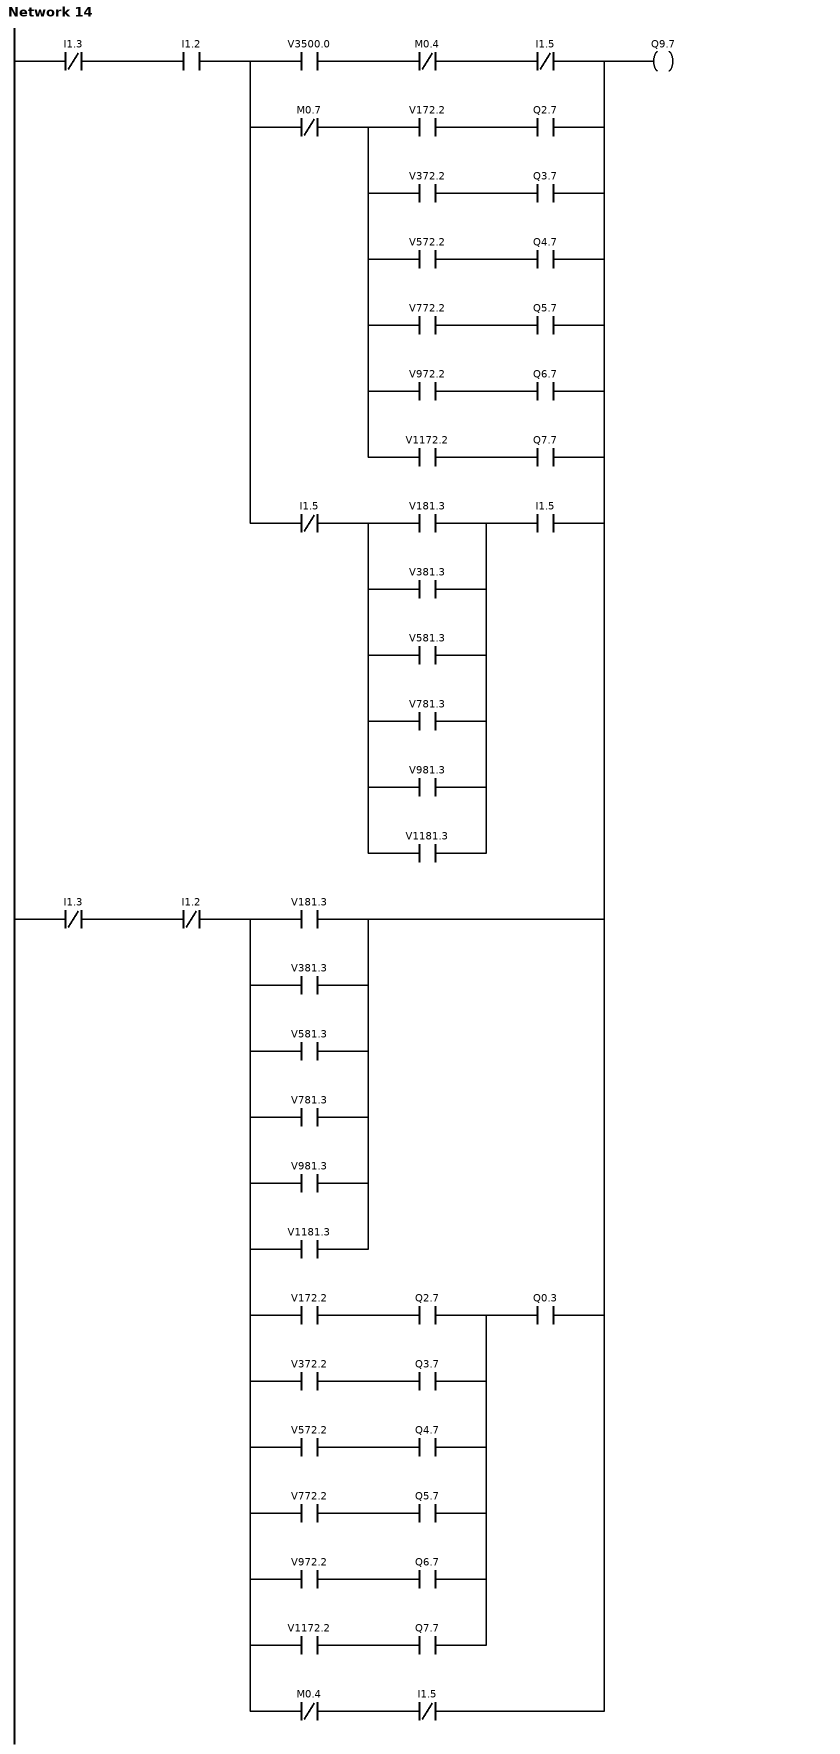
[picture p48: SBR5 networks 14-14]
Network 14
LDN    I1.3
A      I1.2
LD     V3500.0
AN     M0.4
AN     I1.5
LDN    M0.7
LD     V172.2
A      Q2.7
LD     V372.2
A      Q3.7
OLD
LD     V572.2
A      Q4.7
OLD
LD     V772.2
A      Q5.7
OLD
LD     V972.2
A      Q6.7
OLD
LD     V1172.2
A      Q7.7
OLD
ALD
OLD
LDN    I1.5
LD     V181.3
O      V381.3
O      V581.3
O      V781.3
O      V981.3
O      V1181.3
ALD
A      I1.5
OLD
ALD
LDN    I1.3
AN     I1.2
LD     V181.3
O      V381.3
O      V581.3
O      V781.3
O      V981.3
O      V1181.3
LD     V172.2
A      Q2.7
LD     V372.2
A      Q3.7
OLD
LD     V572.2
A      Q4.7
OLD
LD     V772.2
A      Q5.7
OLD
LD     V972.2
A      Q6.7
OLD
LD     V1172.2
A      Q7.7
OLD
A      Q0.3
OLD
LDN    M0.4
AN     I1.5
OLD
ALD
OLD
=      Q9.7
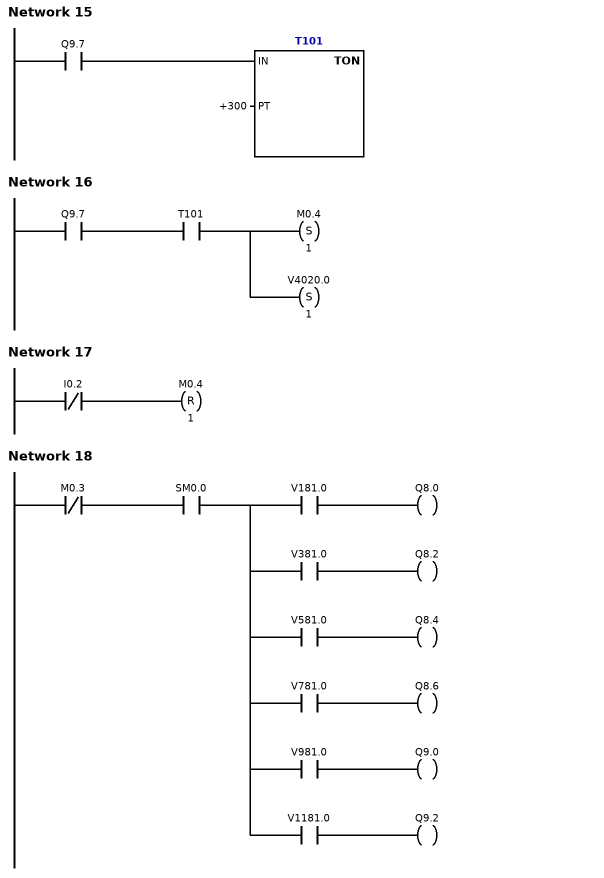
Network 15
LD     Q9.7
TON    T101, +300
Network 16
LD     Q9.7
A      T101
S      M0.4, 1
S      V4020.0, 1
Network 17
LDN    I0.2
R      M0.4, 1
Network 18
LDN    M0.3
A      SM0.0
LPS
A      V181.0
=      Q8.0
LRD
A      V381.0
=      Q8.2
LRD
A      V581.0
=      Q8.4
LRD
A      V781.0
=      Q8.6
LRD
A      V981.0
=      Q9.0
LPP
A      V1181.0
=      Q9.2
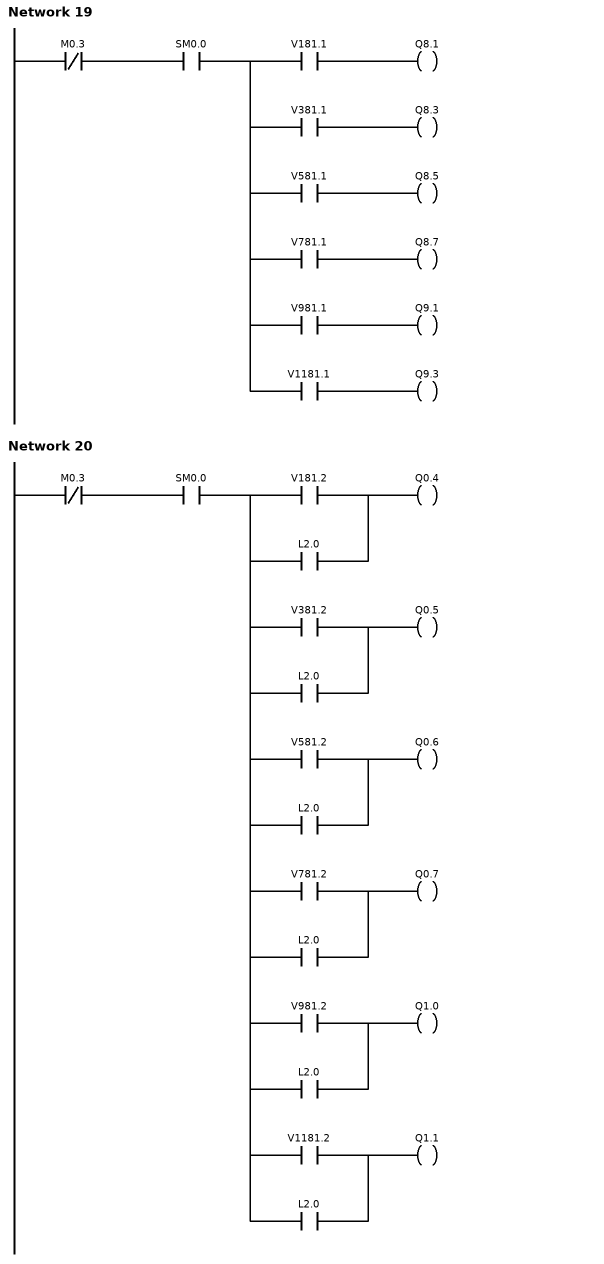
Network 19
LDN    M0.3
A      SM0.0
LPS
A      V181.1
=      Q8.1
LRD
A      V381.1
=      Q8.3
LRD
A      V581.1
=      Q8.5
LRD
A      V781.1
=      Q8.7
LRD
A      V981.1
=      Q9.1
LPP
A      V1181.1
=      Q9.3
Network 20
LDN    M0.3
A      SM0.0
LPS
LD     V181.2
O      L2.0
ALD
=      Q0.4
LRD
LD     V381.2
O      L2.0
ALD
=      Q0.5
LRD
LD     V581.2
O      L2.0
ALD
=      Q0.6
LRD
LD     V781.2
O      L2.0
ALD
=      Q0.7
LRD
LD     V981.2
O      L2.0
ALD
=      Q1.0
LPP
LD     V1181.2
O      L2.0
ALD
=      Q1.1
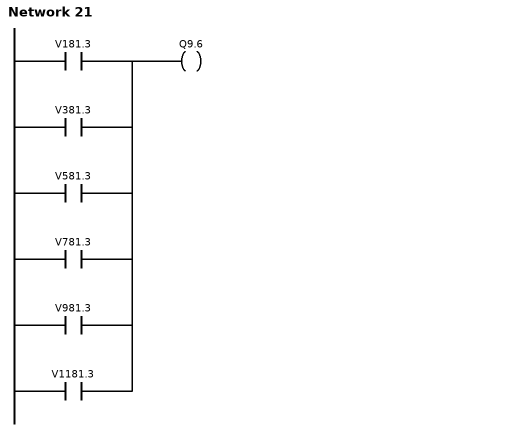
Network 21
LD     V181.3
O      V381.3
O      V581.3
O      V781.3
O      V981.3
O      V1181.3
=      Q9.6
END_SUBROUTINE_BLOCK

SUBROUTINE_BLOCK yz_mc_set:SBR6
TITLE=
BEGIN
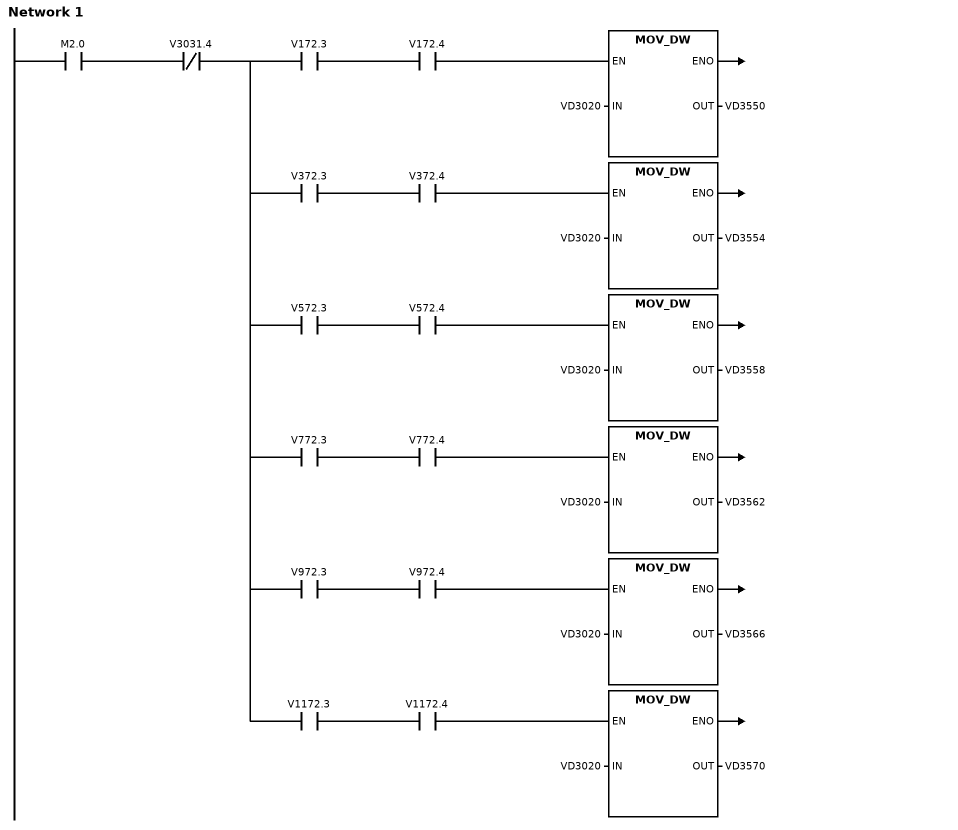
Network 1
LD     M2.0
AN     V3031.4
LPS
A      V172.3
A      V172.4
MOVD   VD3020, VD3550
LRD
A      V372.3
A      V372.4
MOVD   VD3020, VD3554
LRD
A      V572.3
A      V572.4
MOVD   VD3020, VD3558
LRD
A      V772.3
A      V772.4
MOVD   VD3020, VD3562
LRD
A      V972.3
A      V972.4
MOVD   VD3020, VD3566
LPP
A      V1172.3
A      V1172.4
MOVD   VD3020, VD3570
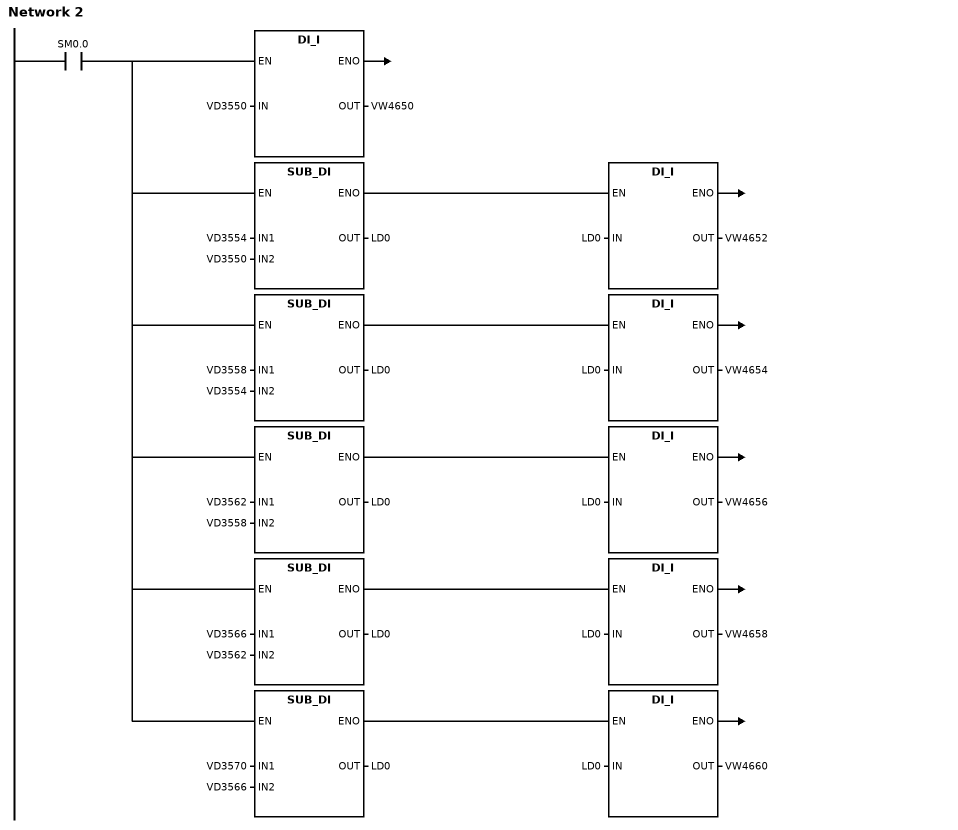
Network 2
LD     SM0.0
LPS
DTI    VD3550, VW4650
MOVD   VD3554, LD0
AENO
-D     VD3550, LD0
AENO
DTI    LD0, VW4652
LRD
MOVD   VD3558, LD0
AENO
-D     VD3554, LD0
AENO
DTI    LD0, VW4654
LRD
MOVD   VD3562, LD0
AENO
-D     VD3558, LD0
AENO
DTI    LD0, VW4656
LRD
MOVD   VD3566, LD0
AENO
-D     VD3562, LD0
AENO
DTI    LD0, VW4658
LPP
MOVD   VD3570, LD0
AENO
-D     VD3566, LD0
AENO
DTI    LD0, VW4660
END_SUBROUTINE_BLOCK

SUBROUTINE_BLOCK STATION_POS:SBR7
TITLE=
BEGIN
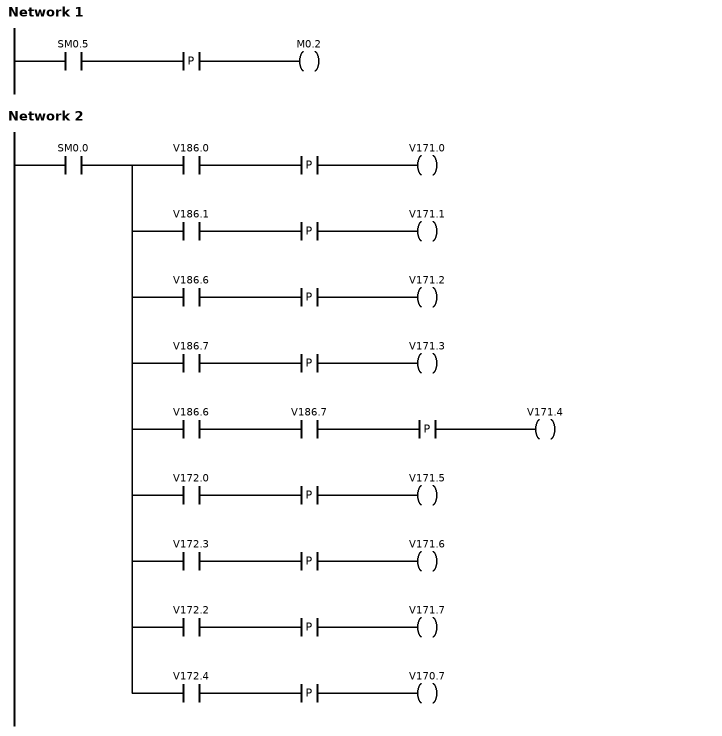
Network 1
LD     SM0.5
EU
=      M0.2
Network 2
LD     SM0.0
LPS
A      V186.0
EU
=      V171.0
LRD
A      V186.1
EU
=      V171.1
LRD
A      V186.6
EU
=      V171.2
LRD
A      V186.7
EU
=      V171.3
LRD
A      V186.6
A      V186.7
EU
=      V171.4
LRD
A      V172.0
EU
=      V171.5
LRD
A      V172.3
EU
=      V171.6
LRD
A      V172.2
EU
=      V171.7
LPP
A      V172.4
EU
=      V170.7
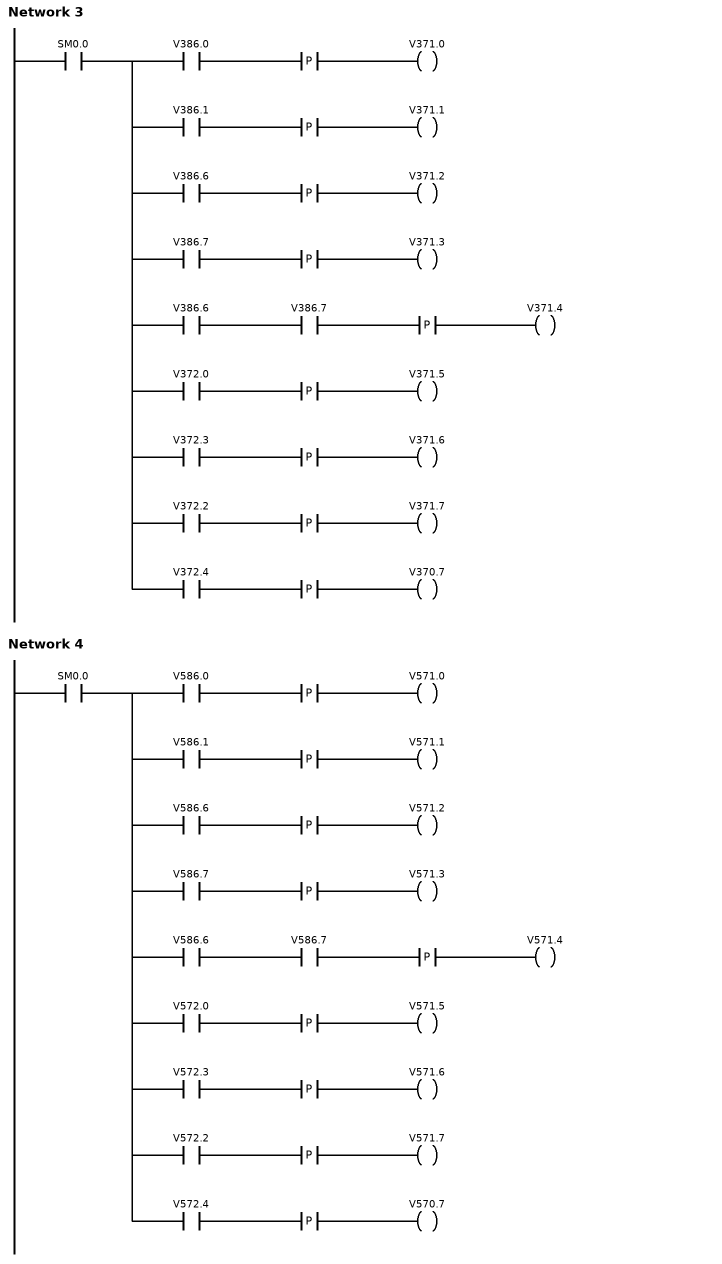
Network 3
LD     SM0.0
LPS
A      V386.0
EU
=      V371.0
LRD
A      V386.1
EU
=      V371.1
LRD
A      V386.6
EU
=      V371.2
LRD
A      V386.7
EU
=      V371.3
LRD
A      V386.6
A      V386.7
EU
=      V371.4
LRD
A      V372.0
EU
=      V371.5
LRD
A      V372.3
EU
=      V371.6
LRD
A      V372.2
EU
=      V371.7
LPP
A      V372.4
EU
=      V370.7
Network 4
LD     SM0.0
LPS
A      V586.0
EU
=      V571.0
LRD
A      V586.1
EU
=      V571.1
LRD
A      V586.6
EU
=      V571.2
LRD
A      V586.7
EU
=      V571.3
LRD
A      V586.6
A      V586.7
EU
=      V571.4
LRD
A      V572.0
EU
=      V571.5
LRD
A      V572.3
EU
=      V571.6
LRD
A      V572.2
EU
=      V571.7
LPP
A      V572.4
EU
=      V570.7
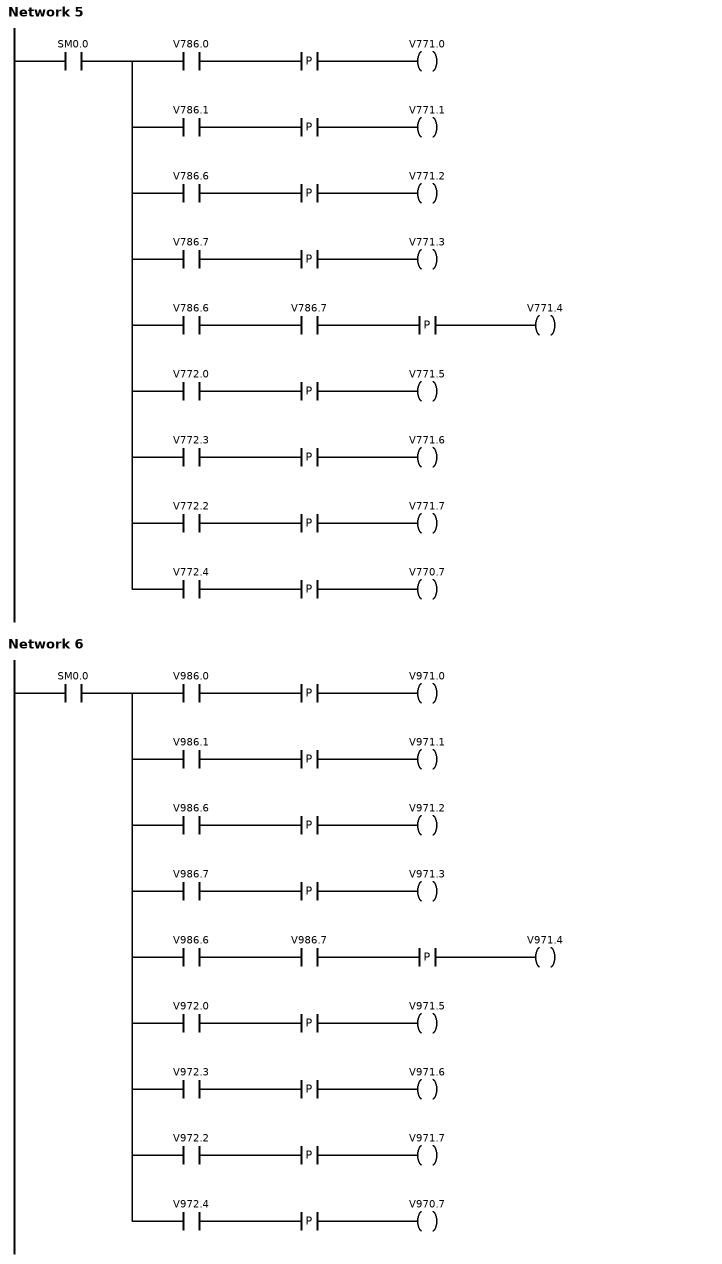
Network 5
LD     SM0.0
LPS
A      V786.0
EU
=      V771.0
LRD
A      V786.1
EU
=      V771.1
LRD
A      V786.6
EU
=      V771.2
LRD
A      V786.7
EU
=      V771.3
LRD
A      V786.6
A      V786.7
EU
=      V771.4
LRD
A      V772.0
EU
=      V771.5
LRD
A      V772.3
EU
=      V771.6
LRD
A      V772.2
EU
=      V771.7
LPP
A      V772.4
EU
=      V770.7
Network 6
LD     SM0.0
LPS
A      V986.0
EU
=      V971.0
LRD
A      V986.1
EU
=      V971.1
LRD
A      V986.6
EU
=      V971.2
LRD
A      V986.7
EU
=      V971.3
LRD
A      V986.6
A      V986.7
EU
=      V971.4
LRD
A      V972.0
EU
=      V971.5
LRD
A      V972.3
EU
=      V971.6
LRD
A      V972.2
EU
=      V971.7
LPP
A      V972.4
EU
=      V970.7
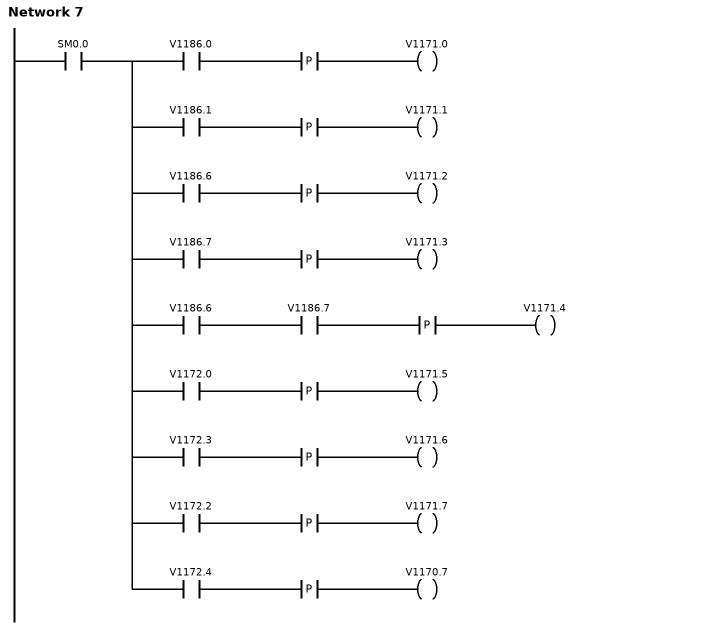
Network 7
LD     SM0.0
LPS
A      V1186.0
EU
=      V1171.0
LRD
A      V1186.1
EU
=      V1171.1
LRD
A      V1186.6
EU
=      V1171.2
LRD
A      V1186.7
EU
=      V1171.3
LRD
A      V1186.6
A      V1186.7
EU
=      V1171.4
LRD
A      V1172.0
EU
=      V1171.5
LRD
A      V1172.3
EU
=      V1171.6
LRD
A      V1172.2
EU
=      V1171.7
LPP
A      V1172.4
EU
=      V1170.7
END_SUBROUTINE_BLOCK

SUBROUTINE_BLOCK AQM_CONTROL:SBR8
TITLE=
BEGIN
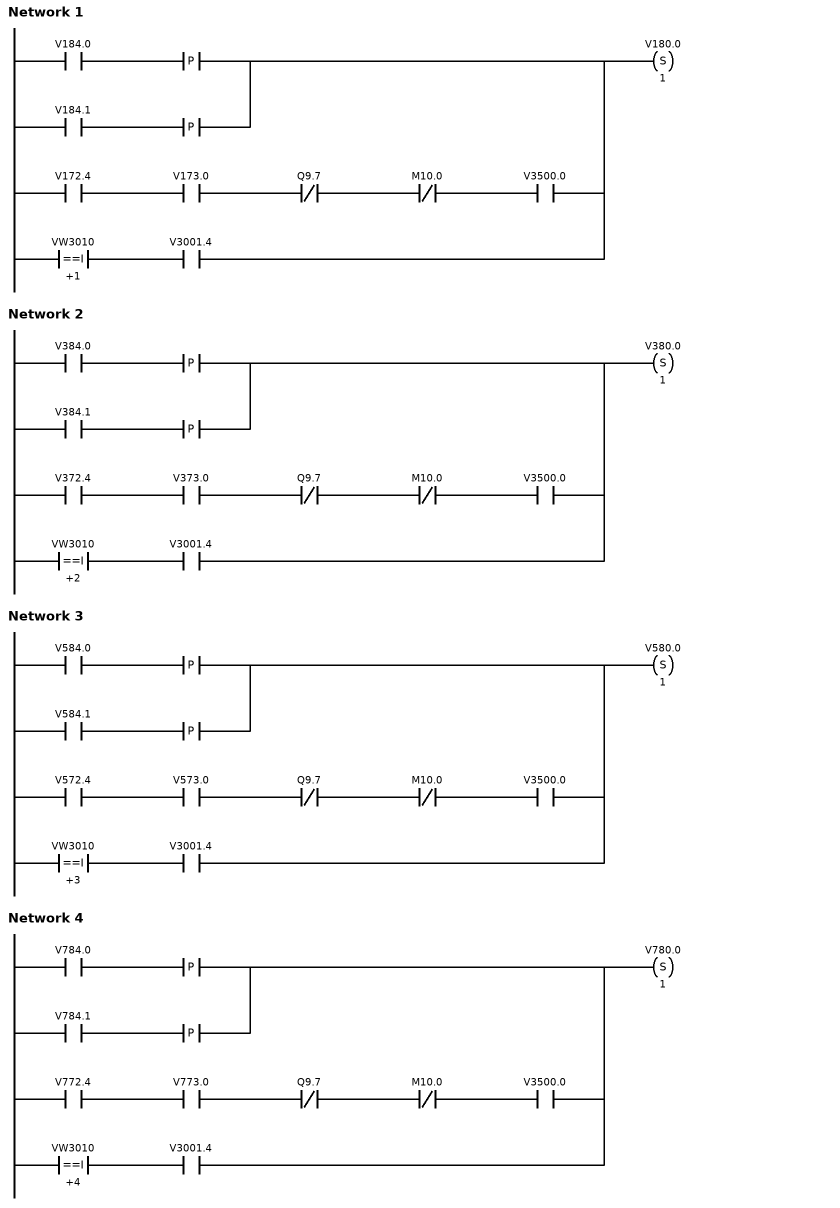
Network 1
LD     V184.0
EU
LD     V184.1
EU
OLD
LD     V172.4
A      V173.0
AN     Q9.7
AN     M10.0
A      V3500.0
OLD
LDW=   VW3010, +1
A      V3001.4
OLD
S      V180.0, 1
Network 2
LD     V384.0
EU
LD     V384.1
EU
OLD
LD     V372.4
A      V373.0
AN     Q9.7
AN     M10.0
A      V3500.0
OLD
LDW=   VW3010, +2
A      V3001.4
OLD
S      V380.0, 1
Network 3
LD     V584.0
EU
LD     V584.1
EU
OLD
LD     V572.4
A      V573.0
AN     Q9.7
AN     M10.0
A      V3500.0
OLD
LDW=   VW3010, +3
A      V3001.4
OLD
S      V580.0, 1
Network 4
LD     V784.0
EU
LD     V784.1
EU
OLD
LD     V772.4
A      V773.0
AN     Q9.7
AN     M10.0
A      V3500.0
OLD
LDW=   VW3010, +4
A      V3001.4
OLD
S      V780.0, 1
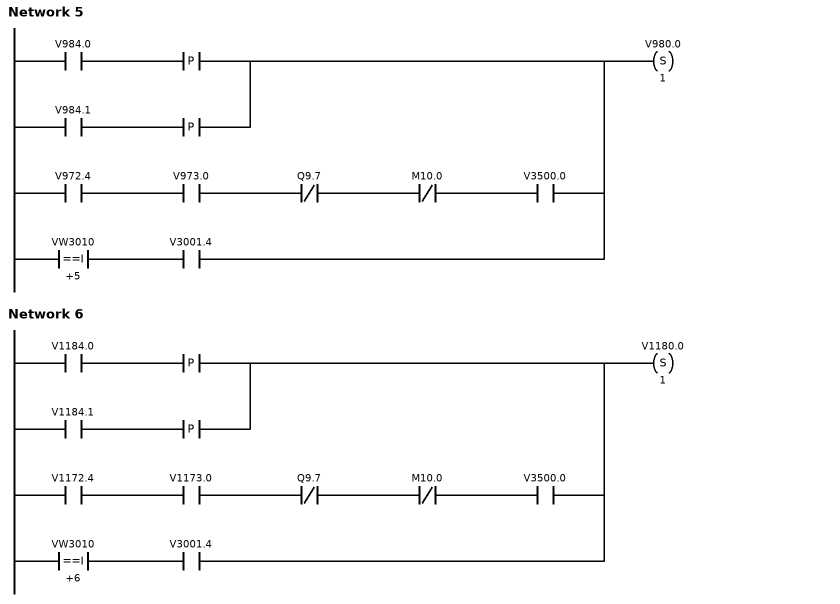
Network 5
LD     V984.0
EU
LD     V984.1
EU
OLD
LD     V972.4
A      V973.0
AN     Q9.7
AN     M10.0
A      V3500.0
OLD
LDW=   VW3010, +5
A      V3001.4
OLD
S      V980.0, 1
Network 6
LD     V1184.0
EU
LD     V1184.1
EU
OLD
LD     V1172.4
A      V1173.0
AN     Q9.7
AN     M10.0
A      V3500.0
OLD
LDW=   VW3010, +6
A      V3001.4
OLD
S      V1180.0, 1
END_SUBROUTINE_BLOCK

SUBROUTINE_BLOCK data_limited:SBR9
TITLE=
BEGIN
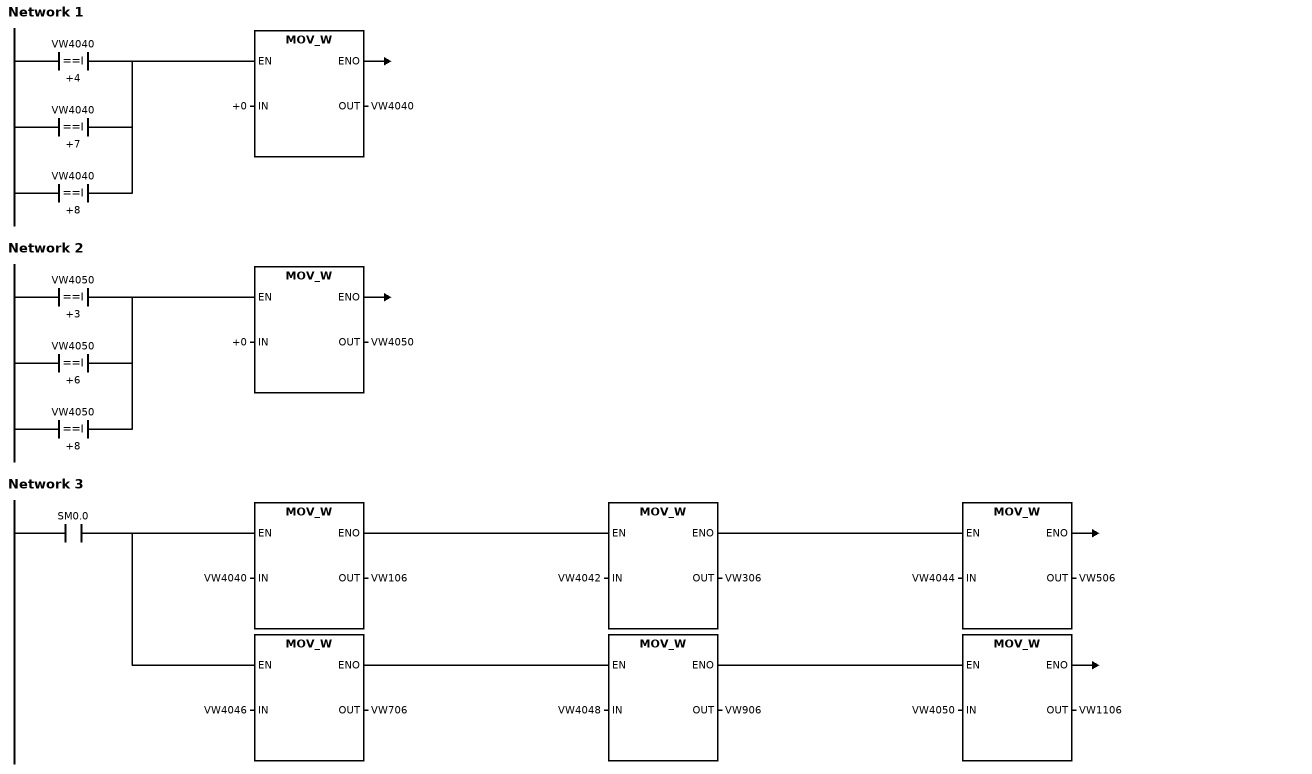
Network 1
LDW=   VW4040, +4
OW=    VW4040, +7
OW=    VW4040, +8
MOVW   +0, VW4040
Network 2
LDW=   VW4050, +3
OW=    VW4050, +6
OW=    VW4050, +8
MOVW   +0, VW4050
Network 3
LD     SM0.0
LPS
MOVW   VW4040, VW106
AENO
MOVW   VW4042, VW306
AENO
MOVW   VW4044, VW506
LPP
MOVW   VW4046, VW706
AENO
MOVW   VW4048, VW906
AENO
MOVW   VW4050, VW1106
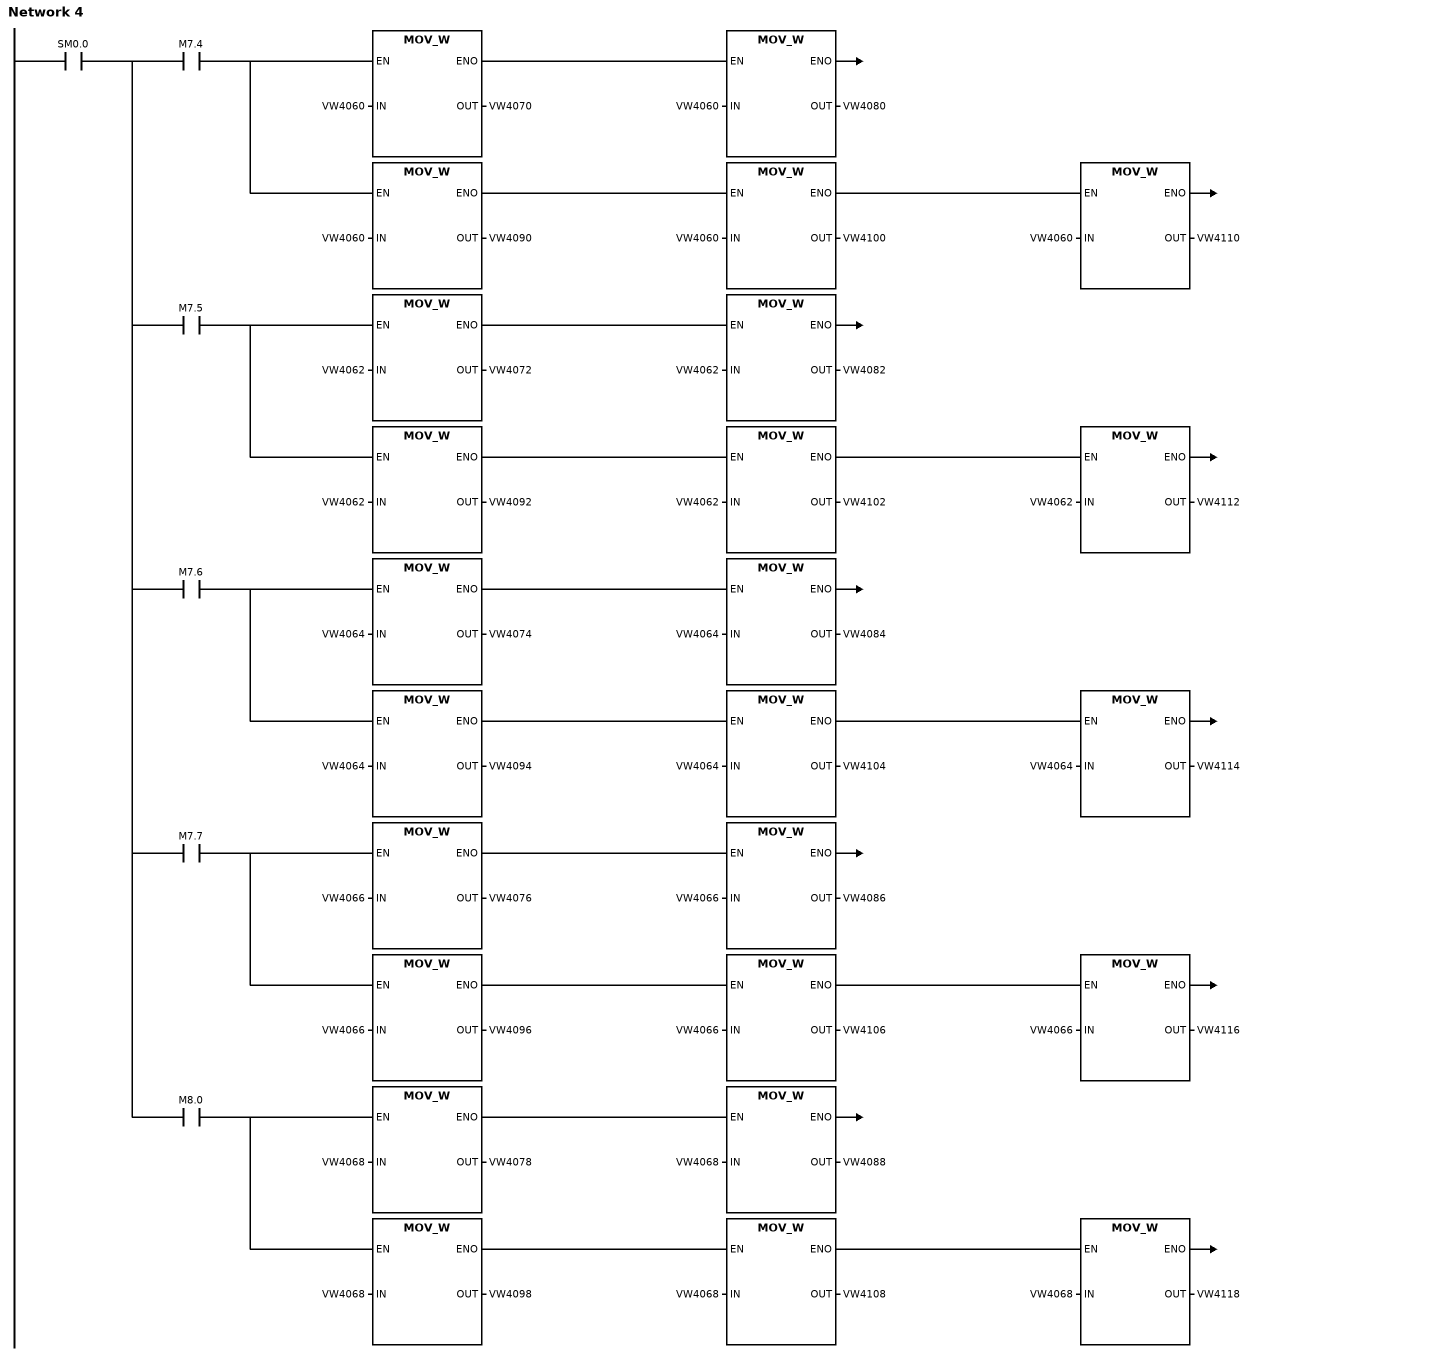
Network 4
LD     SM0.0
LPS
A      M7.4
LPS
MOVW   VW4060, VW4070
AENO
MOVW   VW4060, VW4080
LPP
MOVW   VW4060, VW4090
AENO
MOVW   VW4060, VW4100
AENO
MOVW   VW4060, VW4110
LRD
A      M7.5
LPS
MOVW   VW4062, VW4072
AENO
MOVW   VW4062, VW4082
LPP
MOVW   VW4062, VW4092
AENO
MOVW   VW4062, VW4102
AENO
MOVW   VW4062, VW4112
LRD
A      M7.6
LPS
MOVW   VW4064, VW4074
AENO
MOVW   VW4064, VW4084
LPP
MOVW   VW4064, VW4094
AENO
MOVW   VW4064, VW4104
AENO
MOVW   VW4064, VW4114
LRD
A      M7.7
LPS
MOVW   VW4066, VW4076
AENO
MOVW   VW4066, VW4086
LPP
MOVW   VW4066, VW4096
AENO
MOVW   VW4066, VW4106
AENO
MOVW   VW4066, VW4116
LPP
A      M8.0
LPS
MOVW   VW4068, VW4078
AENO
MOVW   VW4068, VW4088
LPP
MOVW   VW4068, VW4098
AENO
MOVW   VW4068, VW4108
AENO
MOVW   VW4068, VW4118
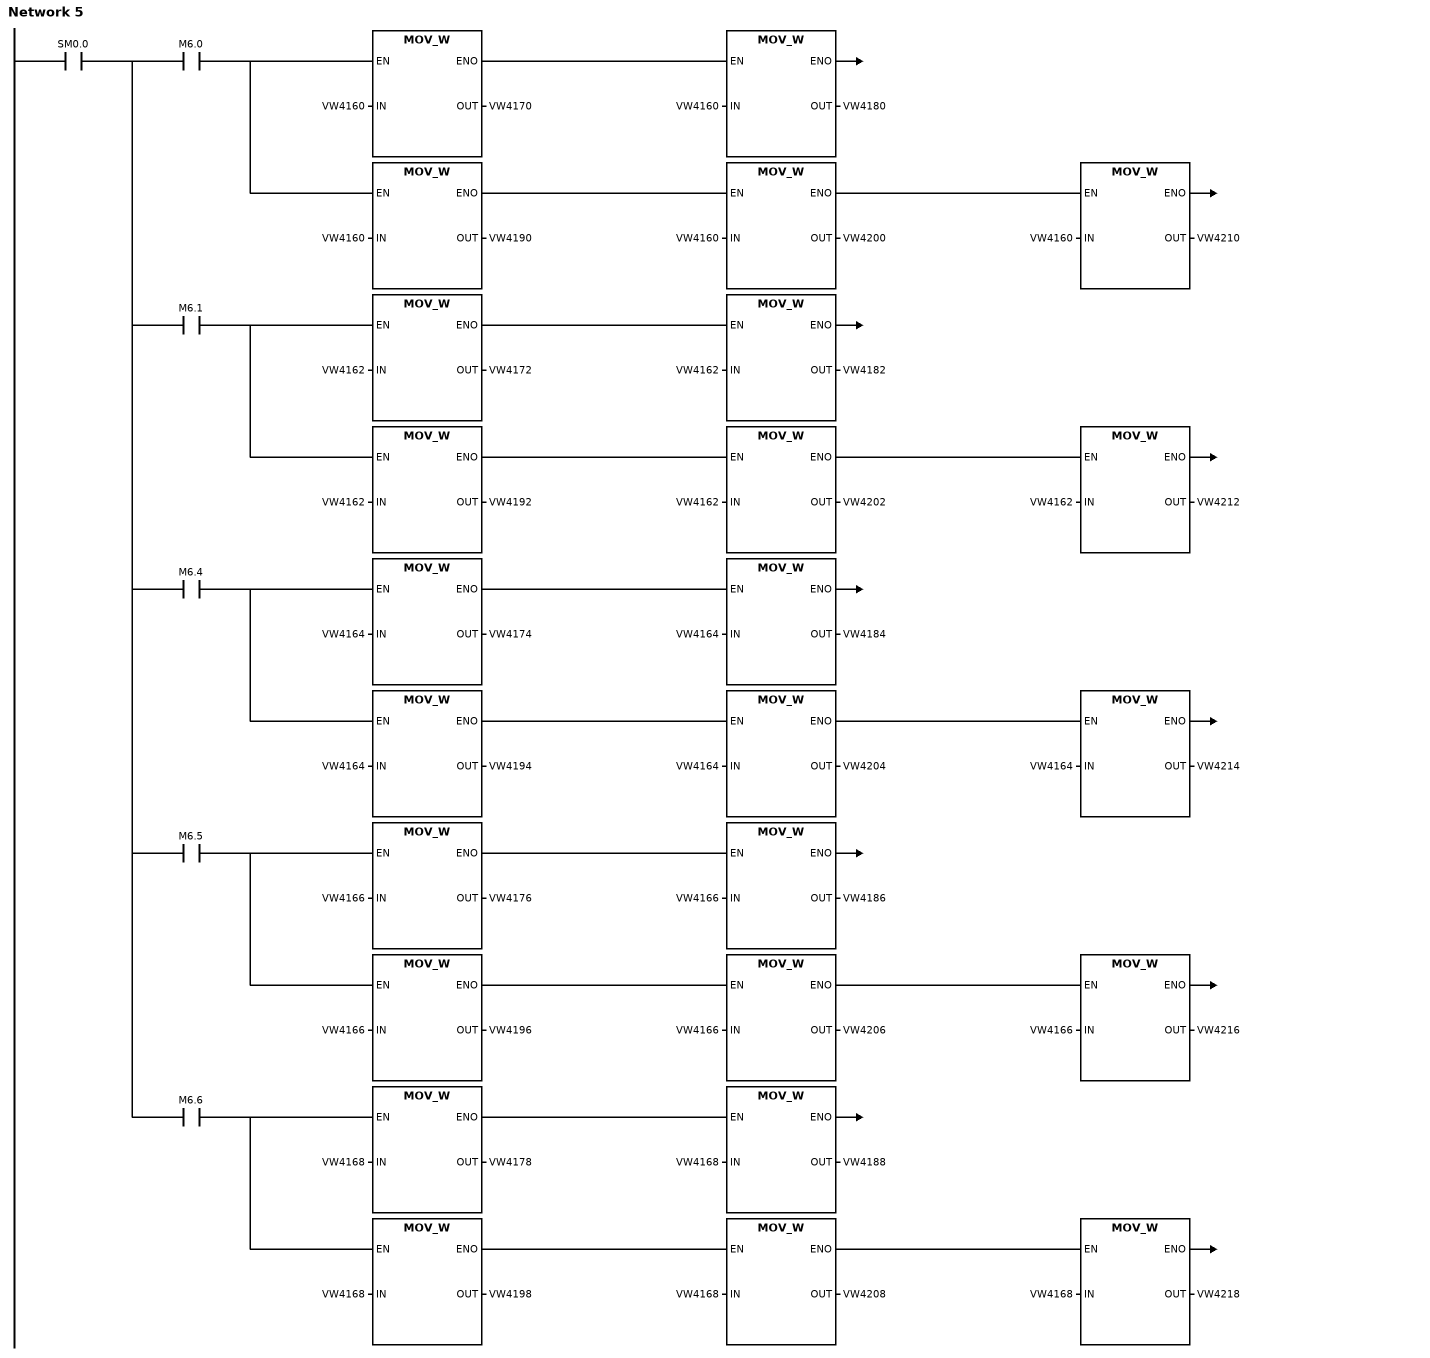
Network 5
LD     SM0.0
LPS
A      M6.0
LPS
MOVW   VW4160, VW4170
AENO
MOVW   VW4160, VW4180
LPP
MOVW   VW4160, VW4190
AENO
MOVW   VW4160, VW4200
AENO
MOVW   VW4160, VW4210
LRD
A      M6.1
LPS
MOVW   VW4162, VW4172
AENO
MOVW   VW4162, VW4182
LPP
MOVW   VW4162, VW4192
AENO
MOVW   VW4162, VW4202
AENO
MOVW   VW4162, VW4212
LRD
A      M6.4
LPS
MOVW   VW4164, VW4174
AENO
MOVW   VW4164, VW4184
LPP
MOVW   VW4164, VW4194
AENO
MOVW   VW4164, VW4204
AENO
MOVW   VW4164, VW4214
LRD
A      M6.5
LPS
MOVW   VW4166, VW4176
AENO
MOVW   VW4166, VW4186
LPP
MOVW   VW4166, VW4196
AENO
MOVW   VW4166, VW4206
AENO
MOVW   VW4166, VW4216
LPP
A      M6.6
LPS
MOVW   VW4168, VW4178
AENO
MOVW   VW4168, VW4188
LPP
MOVW   VW4168, VW4198
AENO
MOVW   VW4168, VW4208
AENO
MOVW   VW4168, VW4218
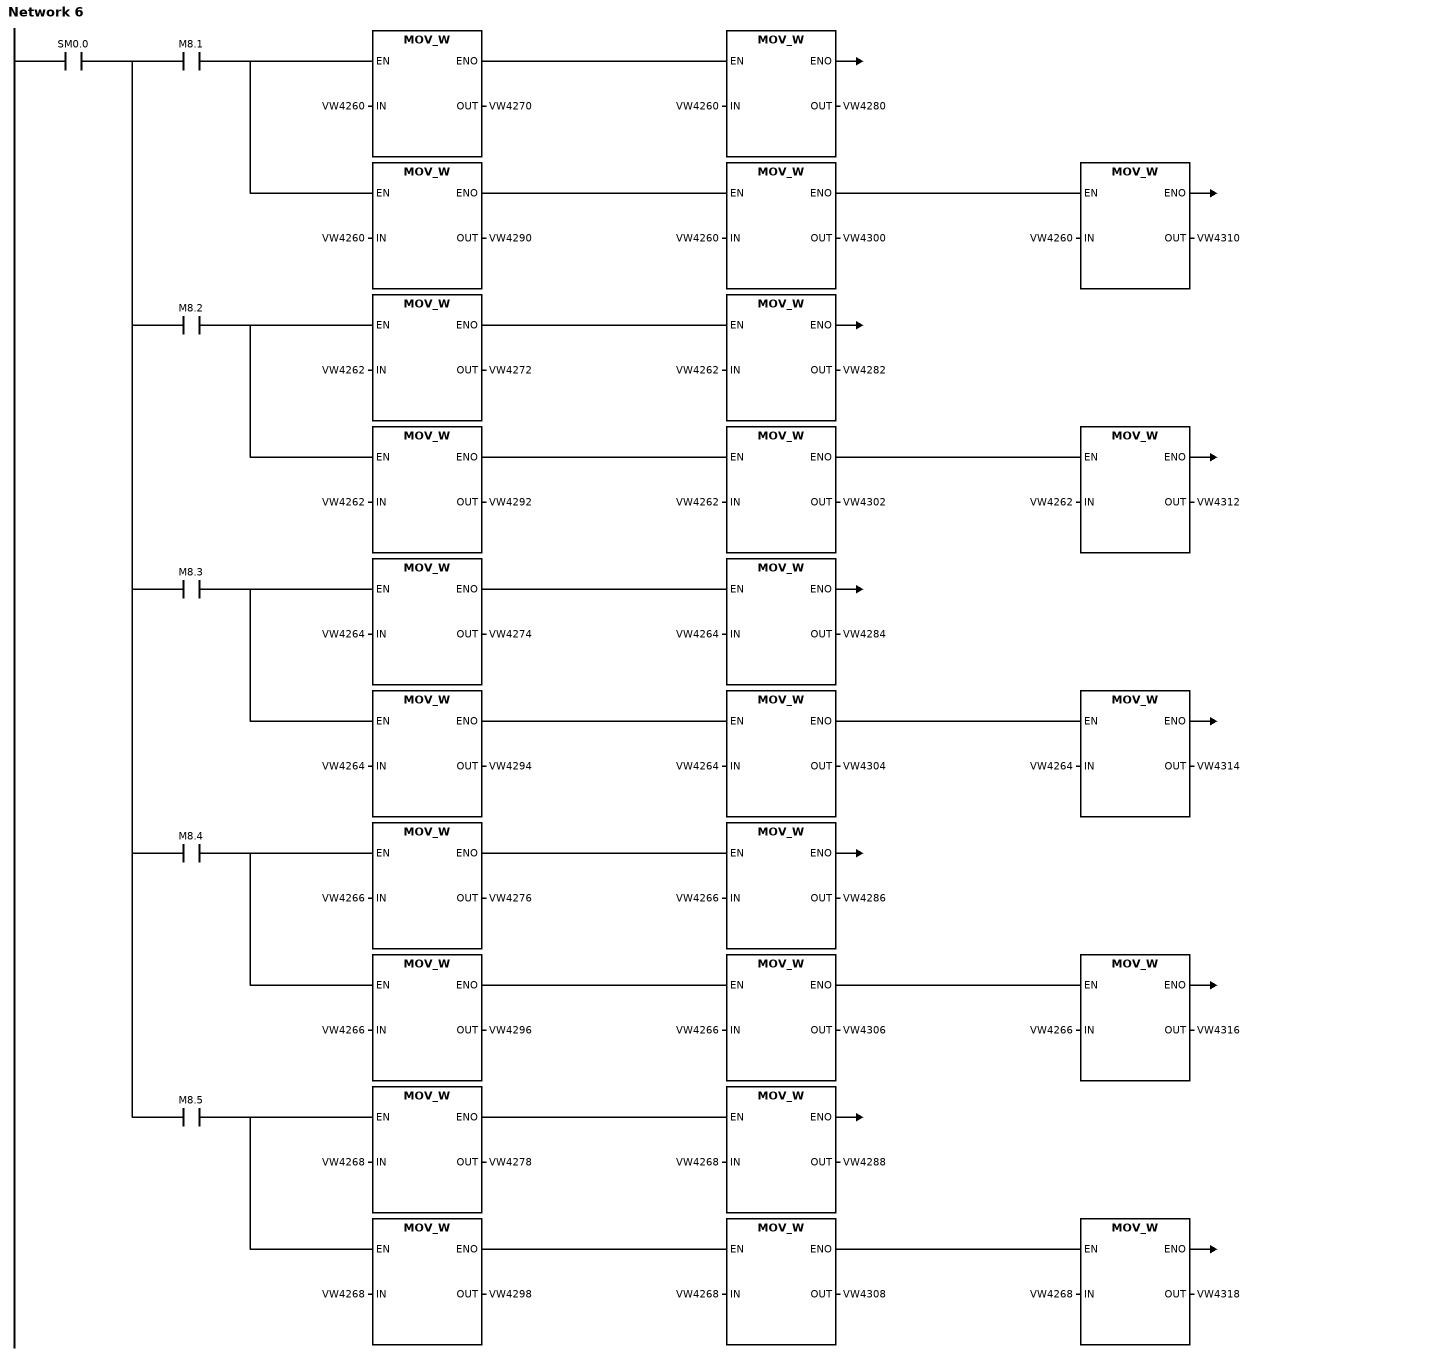
Network 6
LD     SM0.0
LPS
A      M8.1
LPS
MOVW   VW4260, VW4270
AENO
MOVW   VW4260, VW4280
LPP
MOVW   VW4260, VW4290
AENO
MOVW   VW4260, VW4300
AENO
MOVW   VW4260, VW4310
LRD
A      M8.2
LPS
MOVW   VW4262, VW4272
AENO
MOVW   VW4262, VW4282
LPP
MOVW   VW4262, VW4292
AENO
MOVW   VW4262, VW4302
AENO
MOVW   VW4262, VW4312
LRD
A      M8.3
LPS
MOVW   VW4264, VW4274
AENO
MOVW   VW4264, VW4284
LPP
MOVW   VW4264, VW4294
AENO
MOVW   VW4264, VW4304
AENO
MOVW   VW4264, VW4314
LRD
A      M8.4
LPS
MOVW   VW4266, VW4276
AENO
MOVW   VW4266, VW4286
LPP
MOVW   VW4266, VW4296
AENO
MOVW   VW4266, VW4306
AENO
MOVW   VW4266, VW4316
LPP
A      M8.5
LPS
MOVW   VW4268, VW4278
AENO
MOVW   VW4268, VW4288
LPP
MOVW   VW4268, VW4298
AENO
MOVW   VW4268, VW4308
AENO
MOVW   VW4268, VW4318
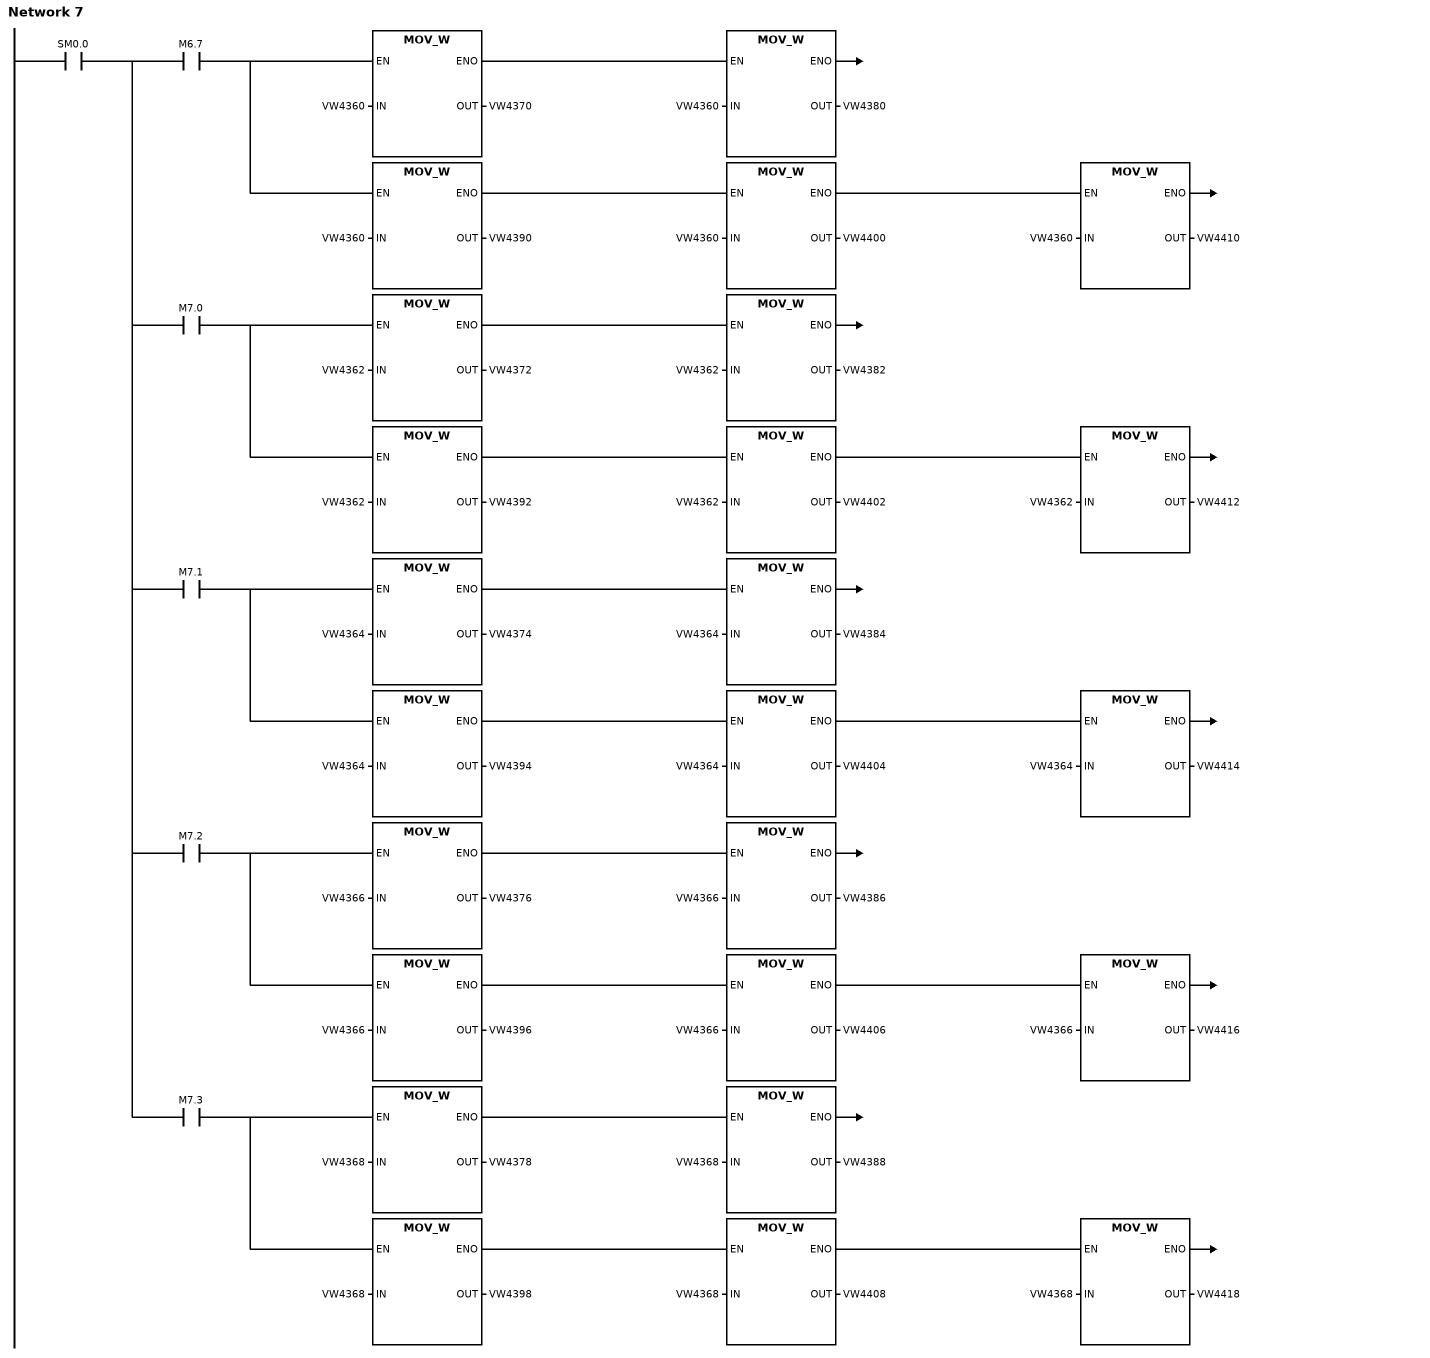
Network 7
LD     SM0.0
LPS
A      M6.7
LPS
MOVW   VW4360, VW4370
AENO
MOVW   VW4360, VW4380
LPP
MOVW   VW4360, VW4390
AENO
MOVW   VW4360, VW4400
AENO
MOVW   VW4360, VW4410
LRD
A      M7.0
LPS
MOVW   VW4362, VW4372
AENO
MOVW   VW4362, VW4382
LPP
MOVW   VW4362, VW4392
AENO
MOVW   VW4362, VW4402
AENO
MOVW   VW4362, VW4412
LRD
A      M7.1
LPS
MOVW   VW4364, VW4374
AENO
MOVW   VW4364, VW4384
LPP
MOVW   VW4364, VW4394
AENO
MOVW   VW4364, VW4404
AENO
MOVW   VW4364, VW4414
LRD
A      M7.2
LPS
MOVW   VW4366, VW4376
AENO
MOVW   VW4366, VW4386
LPP
MOVW   VW4366, VW4396
AENO
MOVW   VW4366, VW4406
AENO
MOVW   VW4366, VW4416
LPP
A      M7.3
LPS
MOVW   VW4368, VW4378
AENO
MOVW   VW4368, VW4388
LPP
MOVW   VW4368, VW4398
AENO
MOVW   VW4368, VW4408
AENO
MOVW   VW4368, VW4418
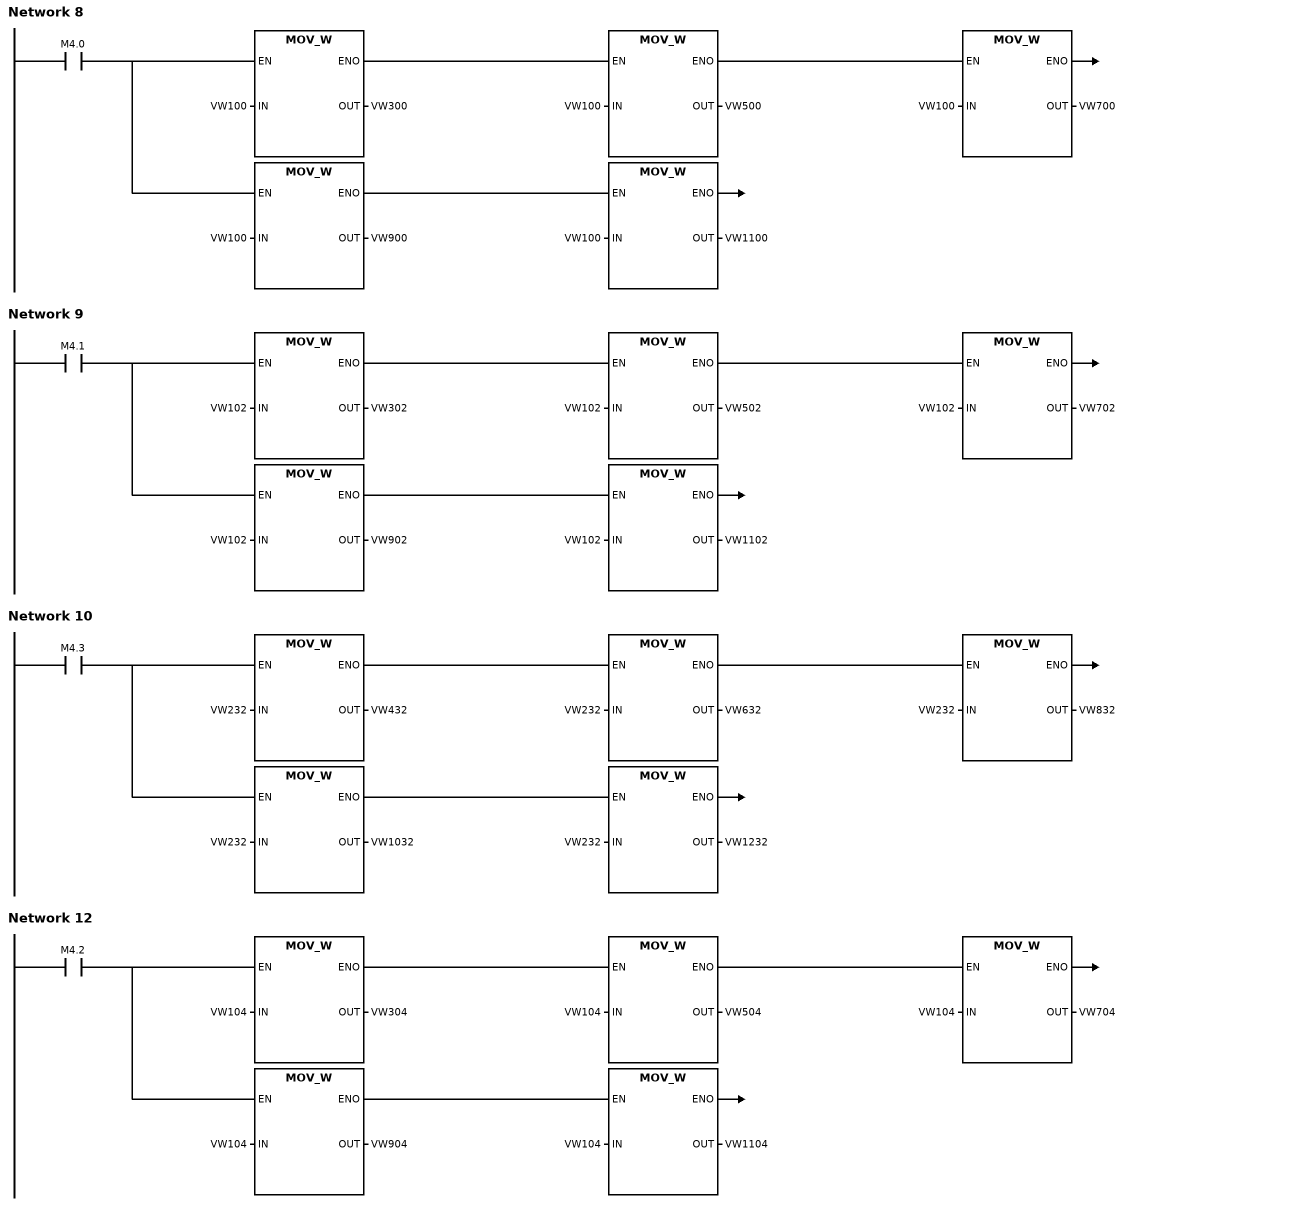
Network 8
LD     M4.0
LPS
MOVW   VW100, VW300
AENO
MOVW   VW100, VW500
AENO
MOVW   VW100, VW700
LPP
MOVW   VW100, VW900
AENO
MOVW   VW100, VW1100
Network 9
LD     M4.1
LPS
MOVW   VW102, VW302
AENO
MOVW   VW102, VW502
AENO
MOVW   VW102, VW702
LPP
MOVW   VW102, VW902
AENO
MOVW   VW102, VW1102
Network 10
LD     M4.3
LPS
MOVW   VW232, VW432
AENO
MOVW   VW232, VW632
AENO
MOVW   VW232, VW832
LPP
MOVW   VW232, VW1032
AENO
MOVW   VW232, VW1232
Network 12
LD     M4.2
LPS
MOVW   VW104, VW304
AENO
MOVW   VW104, VW504
AENO
MOVW   VW104, VW704
LPP
MOVW   VW104, VW904
AENO
MOVW   VW104, VW1104
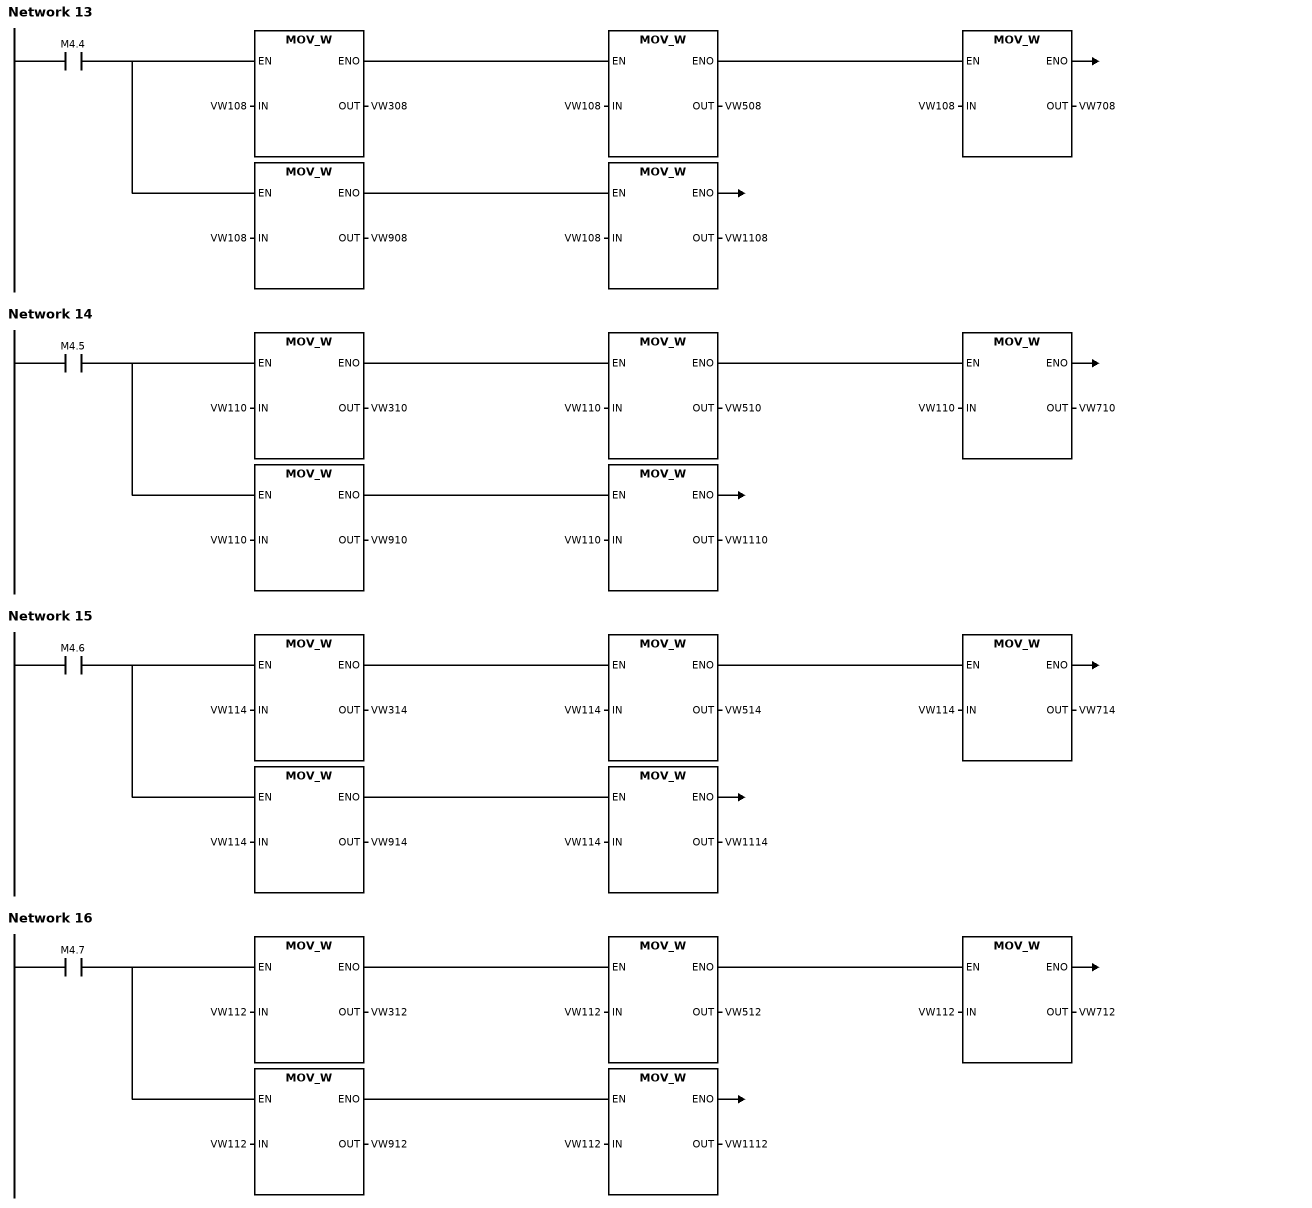
Network 13
LD     M4.4
LPS
MOVW   VW108, VW308
AENO
MOVW   VW108, VW508
AENO
MOVW   VW108, VW708
LPP
MOVW   VW108, VW908
AENO
MOVW   VW108, VW1108
Network 14
LD     M4.5
LPS
MOVW   VW110, VW310
AENO
MOVW   VW110, VW510
AENO
MOVW   VW110, VW710
LPP
MOVW   VW110, VW910
AENO
MOVW   VW110, VW1110
Network 15
LD     M4.6
LPS
MOVW   VW114, VW314
AENO
MOVW   VW114, VW514
AENO
MOVW   VW114, VW714
LPP
MOVW   VW114, VW914
AENO
MOVW   VW114, VW1114
Network 16
LD     M4.7
LPS
MOVW   VW112, VW312
AENO
MOVW   VW112, VW512
AENO
MOVW   VW112, VW712
LPP
MOVW   VW112, VW912
AENO
MOVW   VW112, VW1112
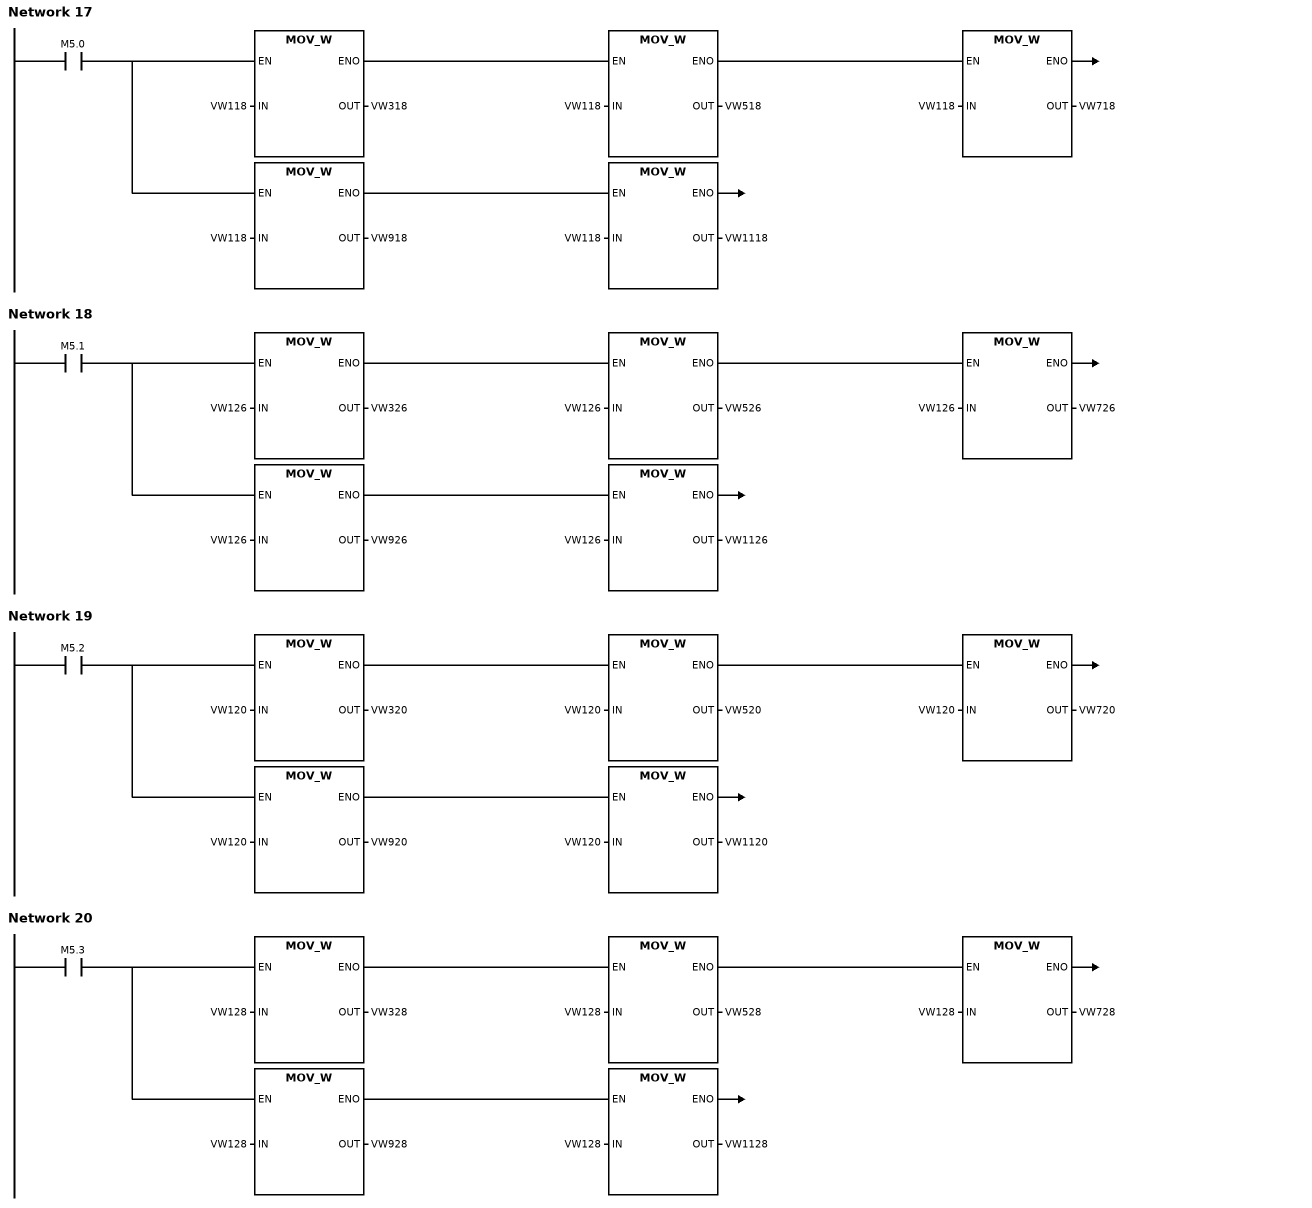
Network 17
LD     M5.0
LPS
MOVW   VW118, VW318
AENO
MOVW   VW118, VW518
AENO
MOVW   VW118, VW718
LPP
MOVW   VW118, VW918
AENO
MOVW   VW118, VW1118
Network 18
LD     M5.1
LPS
MOVW   VW126, VW326
AENO
MOVW   VW126, VW526
AENO
MOVW   VW126, VW726
LPP
MOVW   VW126, VW926
AENO
MOVW   VW126, VW1126
Network 19
LD     M5.2
LPS
MOVW   VW120, VW320
AENO
MOVW   VW120, VW520
AENO
MOVW   VW120, VW720
LPP
MOVW   VW120, VW920
AENO
MOVW   VW120, VW1120
Network 20
LD     M5.3
LPS
MOVW   VW128, VW328
AENO
MOVW   VW128, VW528
AENO
MOVW   VW128, VW728
LPP
MOVW   VW128, VW928
AENO
MOVW   VW128, VW1128
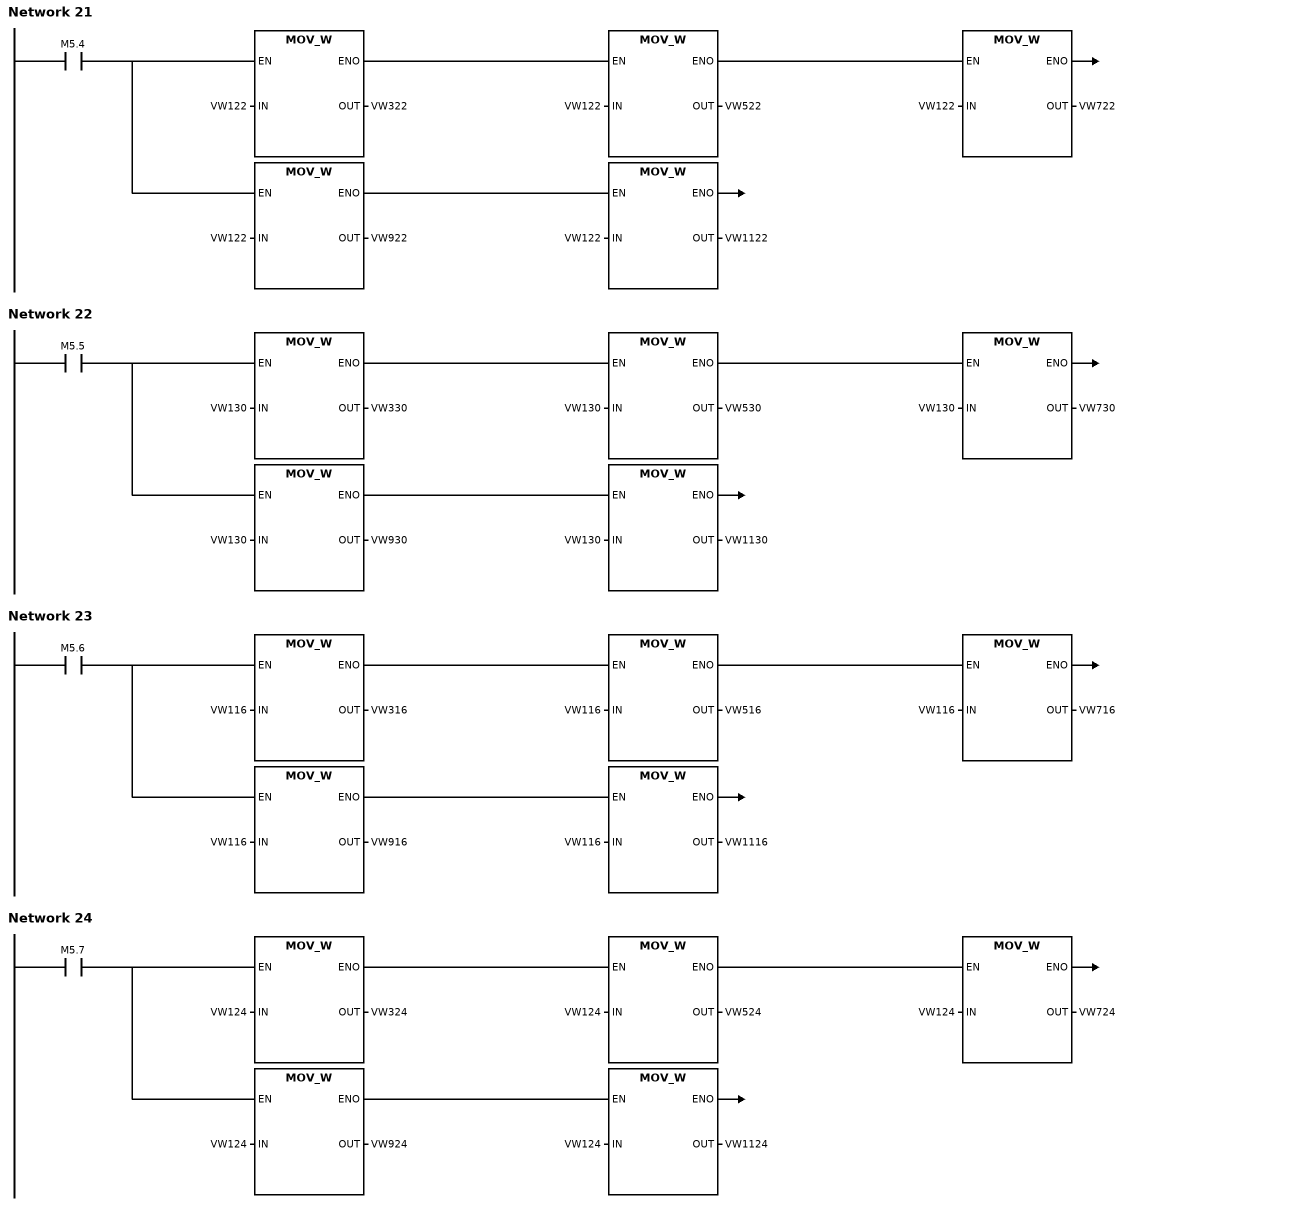
Network 21
LD     M5.4
LPS
MOVW   VW122, VW322
AENO
MOVW   VW122, VW522
AENO
MOVW   VW122, VW722
LPP
MOVW   VW122, VW922
AENO
MOVW   VW122, VW1122
Network 22
LD     M5.5
LPS
MOVW   VW130, VW330
AENO
MOVW   VW130, VW530
AENO
MOVW   VW130, VW730
LPP
MOVW   VW130, VW930
AENO
MOVW   VW130, VW1130
Network 23
LD     M5.6
LPS
MOVW   VW116, VW316
AENO
MOVW   VW116, VW516
AENO
MOVW   VW116, VW716
LPP
MOVW   VW116, VW916
AENO
MOVW   VW116, VW1116
Network 24
LD     M5.7
LPS
MOVW   VW124, VW324
AENO
MOVW   VW124, VW524
AENO
MOVW   VW124, VW724
LPP
MOVW   VW124, VW924
AENO
MOVW   VW124, VW1124
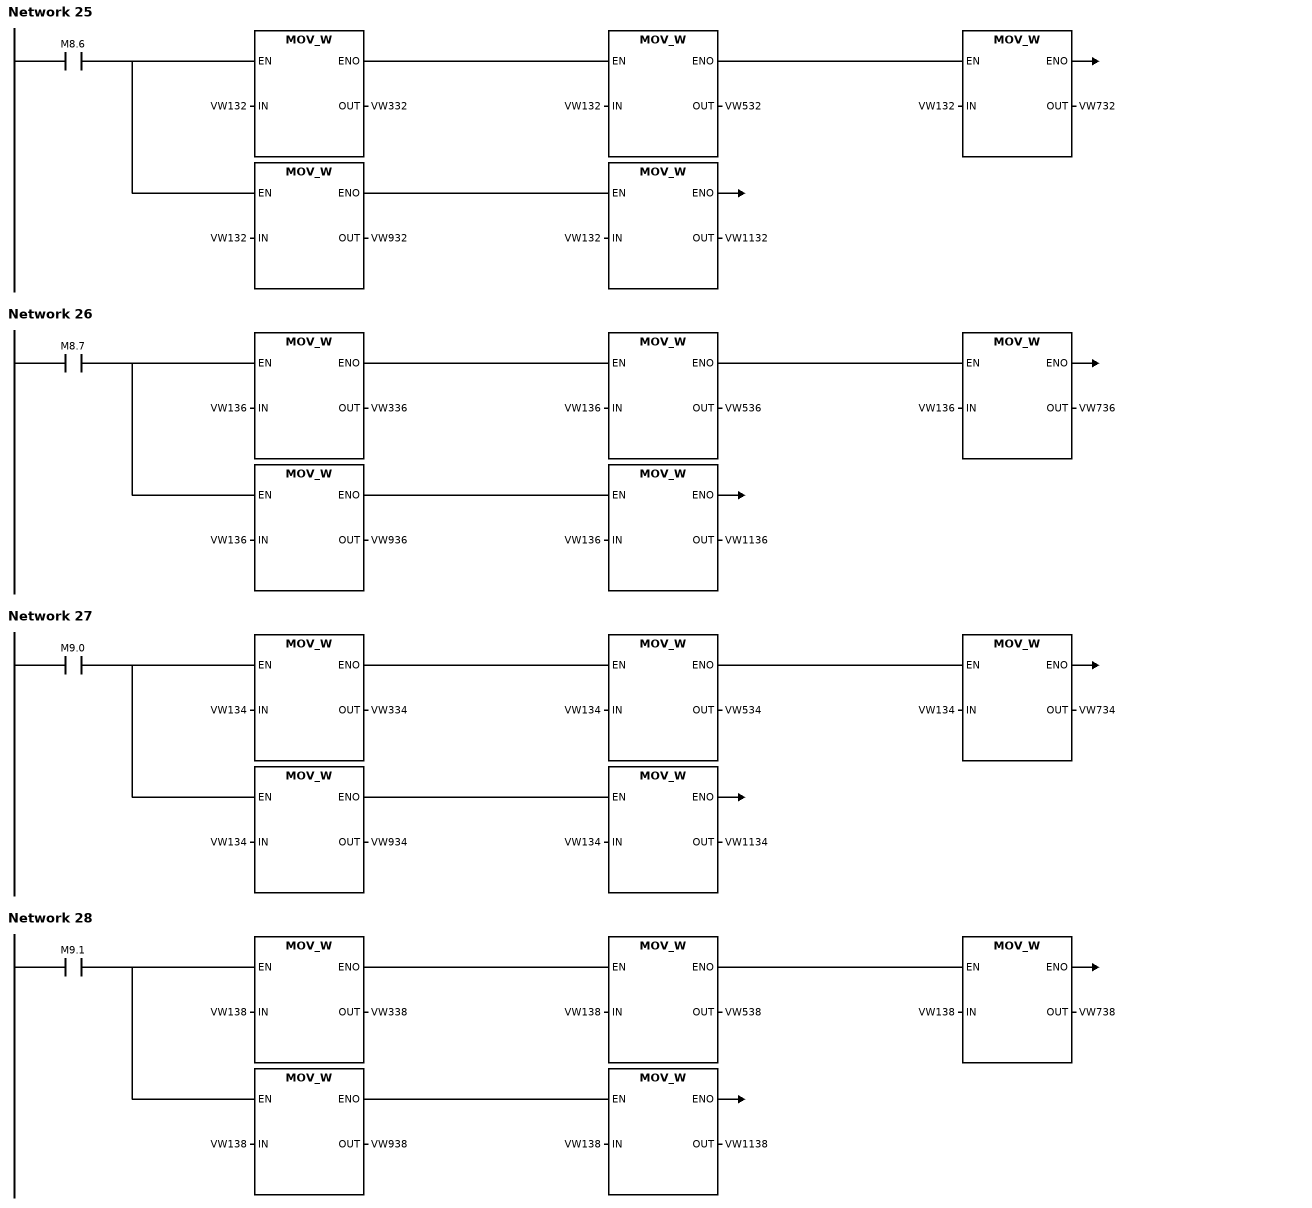
Network 25
LD     M8.6
LPS
MOVW   VW132, VW332
AENO
MOVW   VW132, VW532
AENO
MOVW   VW132, VW732
LPP
MOVW   VW132, VW932
AENO
MOVW   VW132, VW1132
Network 26
LD     M8.7
LPS
MOVW   VW136, VW336
AENO
MOVW   VW136, VW536
AENO
MOVW   VW136, VW736
LPP
MOVW   VW136, VW936
AENO
MOVW   VW136, VW1136
Network 27
LD     M9.0
LPS
MOVW   VW134, VW334
AENO
MOVW   VW134, VW534
AENO
MOVW   VW134, VW734
LPP
MOVW   VW134, VW934
AENO
MOVW   VW134, VW1134
Network 28
LD     M9.1
LPS
MOVW   VW138, VW338
AENO
MOVW   VW138, VW538
AENO
MOVW   VW138, VW738
LPP
MOVW   VW138, VW938
AENO
MOVW   VW138, VW1138
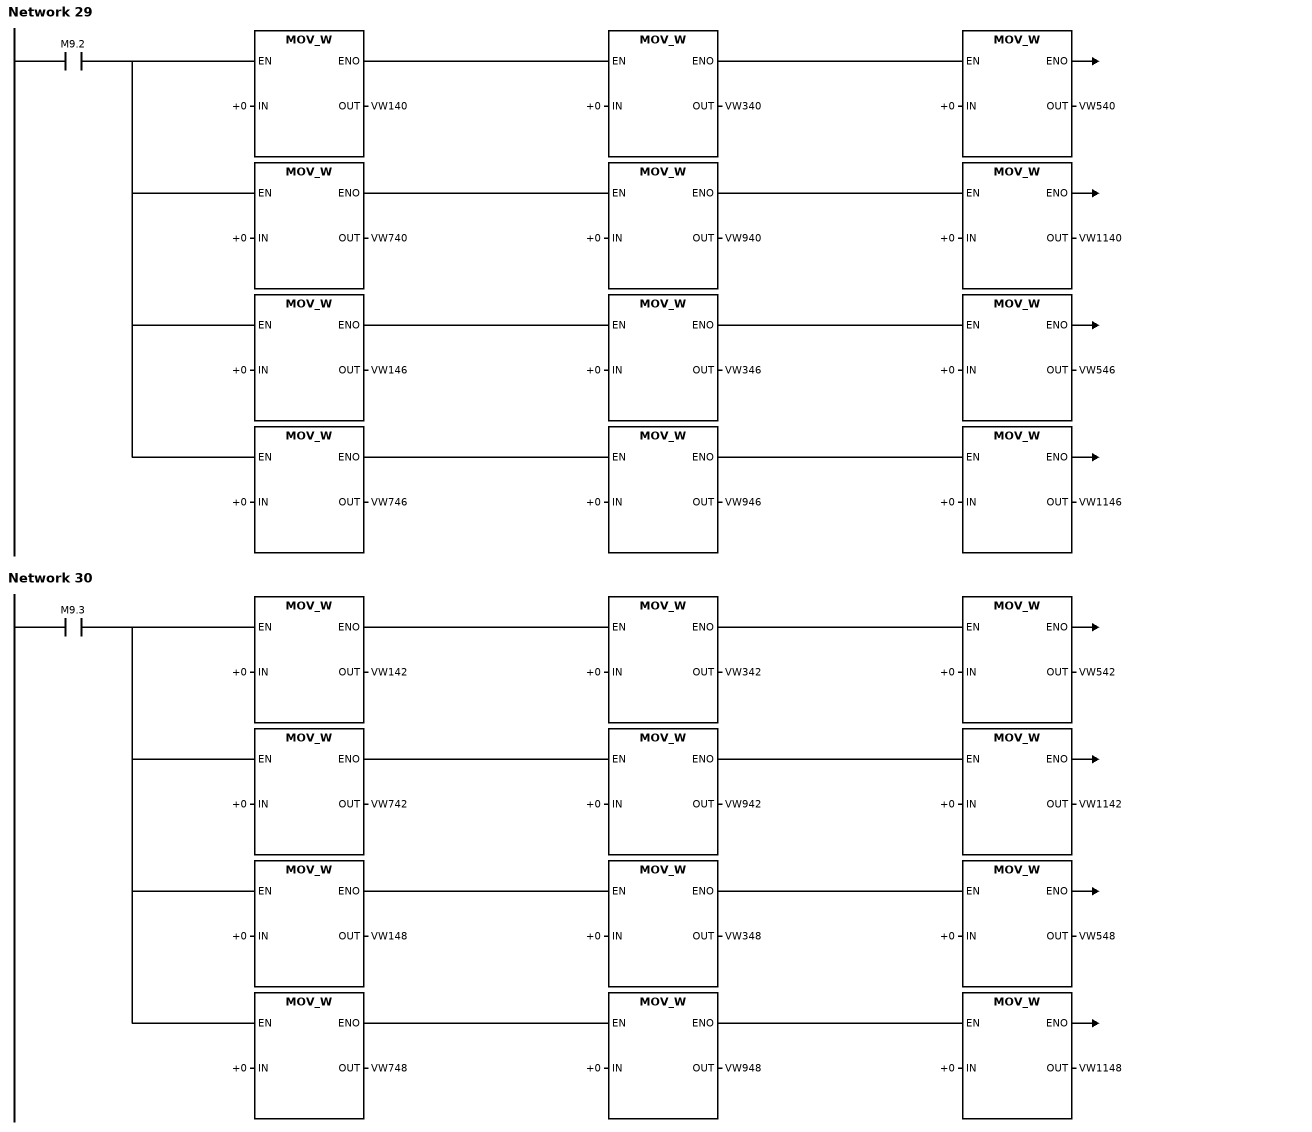
Network 29
LD     M9.2
LPS
MOVW   +0, VW140
AENO
MOVW   +0, VW340
AENO
MOVW   +0, VW540
LRD
MOVW   +0, VW740
AENO
MOVW   +0, VW940
AENO
MOVW   +0, VW1140
LRD
MOVW   +0, VW146
AENO
MOVW   +0, VW346
AENO
MOVW   +0, VW546
LPP
MOVW   +0, VW746
AENO
MOVW   +0, VW946
AENO
MOVW   +0, VW1146
Network 30
LD     M9.3
LPS
MOVW   +0, VW142
AENO
MOVW   +0, VW342
AENO
MOVW   +0, VW542
LRD
MOVW   +0, VW742
AENO
MOVW   +0, VW942
AENO
MOVW   +0, VW1142
LRD
MOVW   +0, VW148
AENO
MOVW   +0, VW348
AENO
MOVW   +0, VW548
LPP
MOVW   +0, VW748
AENO
MOVW   +0, VW948
AENO
MOVW   +0, VW1148
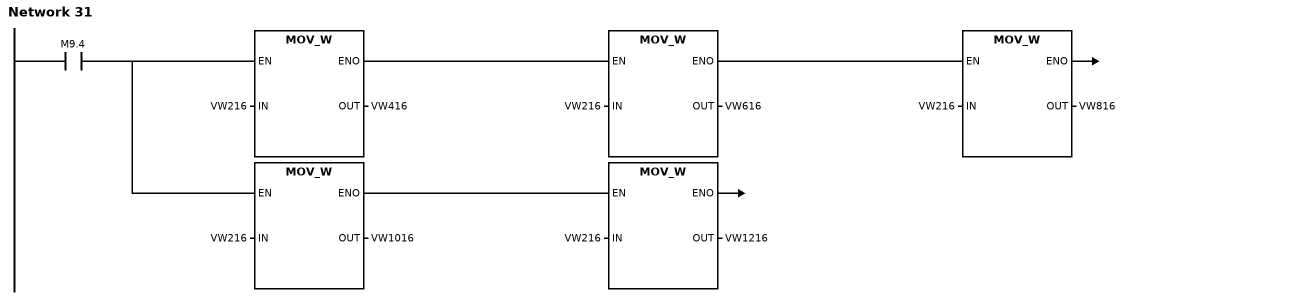
Network 31
LD     M9.4
LPS
MOVW   VW216, VW416
AENO
MOVW   VW216, VW616
AENO
MOVW   VW216, VW816
LPP
MOVW   VW216, VW1016
AENO
MOVW   VW216, VW1216
END_SUBROUTINE_BLOCK

SUBROUTINE_BLOCK data_rcv:SBR10
TITLE=
BEGIN
